Universal Robots PolyScope program: UR_test21122021.urp

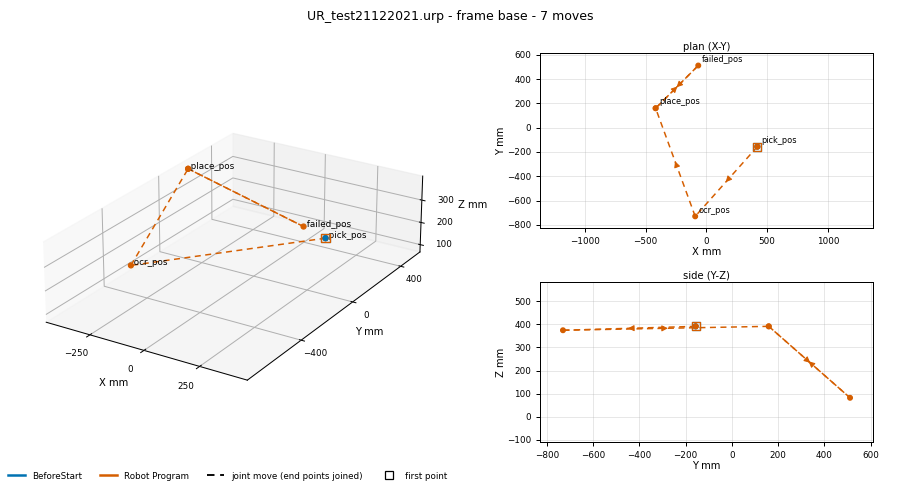
[picture p0: tool path of UR_test21122021.urp in frame base, 7 of 8 moves have a stored position in this frame; points joined in program order, loops and branches not executed]
Program UR_test21122021 (installation=default directory=/programs/test createdIn=3.14.1.1031110 lastSavedIn=3.14.1.1031110 robotSerialNumber=2018300229)
Calibrated DH parameters: a=[-0.000133, -0.610916, -0.569347, 0.000119, -0.000067, 0]; d=[0.127899, 3.644122, -0.017787, -3.463089, 0.115767, 0.092147]; alpha=[1.570708, -0.011279, -0.012231, 1.568854, -1.569164, 0]; deltaTheta=[-0.000097, -0.067195, -0.010506, 0.077758, -0.000102, -0.000058]
BeforeStart
  s_open := socket_open("192.168.0.10",30000)
  MoveJ speed 60 deg/s, acceleration 80 deg/s^2 (useActiveTCP=true)
    Waypoint pick_pos: TCP in base x=419.429 y=-156.467 z=391.085 mm, rx=2.1805 ry=-2.2613 rz=0.0028 rad; joints [0.107, -63.9, -116.333, -89.801, 89.474, 2.62] deg; flange x=419.222 y=-156.192 z=582.085 mm, rx=2.1805 ry=-2.2613 rz=0.0028 rad
  Loop While (checkContinuously=false) expression=s_open ≟  False
    s_open := socket_open("192.168.0.10",30000)
  robot_start := "robot start"
  server_start := "server start"
  part_found := "part found"
  part_n_found := "part not found"
  go_ocr := "go ocr"
  ocr_position := "ocr position"
  part_placed := "part placed"
  go_pick := "go pick"
  var_2 := "0"
Robot Program (runOnlyOnce=false)
  toserver := robot_start
  Script: socket_send_string(toserver)
  Wait Sleep waitTime=0.01
  fromserver := socket_read_string()
  Loop While (checkContinuously=false) expression=fromserver ≠ server_start
    fromserver := socket_read_string()
    Wait Sleep waitTime=0.01
  Folder campos_1
    Loop Forever
      MoveJ speed 60 deg/s, acceleration 80 deg/s^2 (useActiveTCP=true)
        Waypoint pick_pos: motionParameters(blendRadius=0.1); TCP in base x=419.429 y=-156.467 z=391.085 mm, rx=2.1805 ry=-2.2613 rz=0.0028 rad; joints [0.107, -63.9, -116.333, -89.801, 89.474, 2.62] deg; flange x=419.222 y=-156.192 z=582.085 mm, rx=2.1805 ry=-2.2613 rz=0.0028 rad
